Staubli VAL3: Form_PattenD.pgx

public program Form_PattenD(string x_sTitle)
begin
  call Form_PattenS(x_sTitle,"插入,删除,,,,,,,,,退出,,,","F1,F2,F3,F4,F5,F6,F7,F8")
  call Control_PanelD()

end
